PROGRAM MAIN
VAR
//	UpdateEventTimestam : ST_Event;
	aBoolean : BOOL := FALSE;
		
	eEventType1 : E_EventType := E_EventType.Alarm;
	eEventSeverity1 : TcEventSeverity := TcEventSeverity.Error;
	nEventIdentity1 : UDINT := 42;
	sEventText1 : STRING(255) := 'This is a scary event';
	
	CsvPersistentEventStorage : FB_CsvlPersistentEventStorage;
	EventLogger : EventLogger(CsvPersistentEventStorage); // FB_init call leads to error
END_VAR

//IF NOT aBoolean THEN
//	UpdateEventTimestampWithSystemTime(stEvent := UpdateEventTimestam);
//	aBoolean := TRUE;
//END_IF

IF aBoolean THEN
	EventLogger.AddEvent(eEventType1, eEventSeverity1, nEventIdentity1, sEventText1);
	aBoolean := FALSE;
END_IF

CsvPersistentEventStorage();

END_PROGRAM

(* stored: Version 1.1.0.1, ProductVersion 3.1.4024.12
   POU MAIN: Id {d4f3102d-e1ae-4b2b-b4db-93a258302be5}, SpecialFunc None *)
